TEXTLIST MainStateList
  0 = 'Idle'
  1 = 'Disabled'
  2 = 'PreStandby'
  3 = 'Standby'
  4 = 'Manual'
  5 = 'Buffering'
  6 = 'ContinuousExecution'
  7 = 'Fault'
  8 = 'Test'
  9 = 'Recovery'
   = ''
END_TEXTLIST

(* stored: Version 1.1.0.1, ProductVersion 3.1.4024.12
   TextList MainStateList: Id {def977b6-0192-477a-aa92-ed220fcba50e} *)
